PROGRAM Hour_Meter
VAR PERSISTENT
  	MyTimer   : TON;
	TempRun: BOOL;
END_VAR
VAR PERSISTENT
	TotalHours : REAL;
	TotalMinutes : REAL;
END_VAR

MyTimer(IN := TempRun, PT := T#1M);

IF GVL.Pelletizer_Running THEN
	TempRun:= TRUE;
END_IF

IF MyTimer.Q THEN
	TotalMinutes := TotalMinutes + 1;
	TotalHours := TotalHours + (1 / 60);
	TempRun := FALSE;
END_IF


IF TotalMinutes >= 60 THEN
	TotalHours := TotalHours + 1;	
	TotalMinutes := 0;
END_IF

END_PROGRAM

(* stored: Version 1.1.0.1, ProductVersion 3.1.4024.12
   POU Hour_Meter: Id {153ad40f-8882-4e0d-9130-aee4ac2d8039}, SpecialFunc None *)
